// TIA Portal project "FactoryIO_assembler" (V19)
// Vorlageprojekt für das Buch mit Zielsystem S7-1200

(* hardware
DEVICE "S7-1200-Station_1"  S7-1200 Station
   slot 0: "Baugruppenträger_0"  Rack  V1.0
   slot 1: "PLC_1"  CPU 1211C DC/DC/DC  6ES7 211-1AE40-0XB0  V4.1
*)

// ===== PLC "PLC_1"  CPU 1211C DC/DC/DC =====

VAR_GLOBAL   // PLC tag table "Standard-Variablentabelle"
   "Move_X" AT %A0.0 : Bool;
   "Moving_X" AT %E0.0 : Bool;
   "Moving_Z" AT %E0.1 : Bool;
   "FactoryIO_Running" AT %I1.7 : Bool;
   "Start" AT %I1.2 : Bool;
   "Reset" AT %I1.3 : Bool;
   "Stop" AT %I1.4 : Bool;
   "Emergency_Stop" AT %I1.5 : Bool;
   "Auto" AT %I1.6 : Bool;
   "Move_Z" AT %Q0.1 : Bool;
   "Grab" AT %Q0.2 : Bool;
   "Lids_conveyor" AT %Q0.3 : Bool;
   "Clamp_lid" AT %Q0.4 : Bool;
   "Pos_raise" AT %Q0.5 : Bool;
   "Bases_conveyor" AT %Q0.6 : Bool;
   "Start_light" AT %Q1.1 : Bool;
   "Reset light" AT %Q1.2 : Bool;
   "Stop light" AT %Q1.3 : Bool;
   "Counter" AT %QD30 : DInt;
   "Item_detected" AT %I0.2 : Bool;
   "Lid_at_place" AT %I0.3 : Bool;
   "Lid_clamped" AT %I0.4 : Bool;
   "Pos_at_limit (lids)" AT %I0.5 : Bool;
   "Base_at_place" AT %I0.6 : Bool;
   "Base_clamped" AT %I0.7 : Bool;
   "Pos_at_limit (bases)" AT %I1.0 : Bool;
   "Part_leaving" AT %I1.1 : Bool;
   "Clamp_base" AT %Q0.7 : Bool;
   "Pos_raise (bases)" AT %Q1.0 : Bool;
   "Tag_1" AT %M0.0 : Bool;
   "Tag_2" AT %M0.1 : Bool;
   "Tag_3" AT %M0.2 : Bool;
   "Tag_4" AT %M0.3 : Bool;
   "Tag_5" AT %M0.4 : Bool;
   "Tag_6" AT %M0.5 : Bool;
   "Lid_aligned" AT %M0.6 : Bool;
   "Tag_7" AT %M0.7 : Bool;
   "Tag_8" AT %M1.0 : Bool;
   "base_aligned" AT %M1.1 : Bool;
   "Tag_9" AT %M1.2 : Bool;
   "Move_Z_bit" AT %M1.3 : Bool;
   "Tag_10" AT %M1.4 : Bool;
   "Tag_11" AT %M1.5 : Bool;
   "Tag_12" AT %M1.6 : Bool;
   "Tag_13" AT %M1.7 : Bool;
   "Tag_14" AT %M2.0 : Bool;
   "Tag_15" AT %M2.2 : Bool;
   "Move_Z_bit2" AT %M2.1 : Bool;
   "combined_bit" AT %M2.3 : Bool;
   "Tag_16" AT %M2.4 : Bool;
   "Home_bit" AT %M2.5 : Bool;
   "Tag_17" AT %M2.6 : Bool;
END_VAR

// folder: System blocks/Program resources

DATA_BLOCK "IEC_Timer_0_DB"   // DB1
{ S7_Optimized_Access := 'TRUE' }
AUTHOR : Simatic
FAMILY : IEC
NAME : IEC_TMR
VERSION : 1.0
// stored: InstanceOfName IEC_TIMER
"IEC_TIMER"
BEGIN
END_DATA_BLOCK

DATA_BLOCK "IEC_Timer_0_DB_1"   // DB2
{ S7_Optimized_Access := 'TRUE' }
AUTHOR : Simatic
FAMILY : IEC
NAME : IEC_TMR
VERSION : 1.0
// stored: InstanceOfName IEC_TIMER
"IEC_TIMER"
BEGIN
END_DATA_BLOCK

DATA_BLOCK "IEC_Timer_0_DB_2"   // DB3
{ S7_Optimized_Access := 'TRUE' }
AUTHOR : Simatic
FAMILY : IEC
NAME : IEC_TMR
VERSION : 1.0
// stored: InstanceOfName IEC_TIMER
"IEC_TIMER"
BEGIN
END_DATA_BLOCK

// folder: (top level)

FUNCTION "conveyor" : Void   // FC1, LAD
{ S7_Optimized_Access := 'TRUE' }
VERSION : 0.1
   VAR_TEMP   // added for the SCL form of the ladder/FBD networks
      _w1 : Bool;
   END_VAR
BEGIN

REGION Network 1
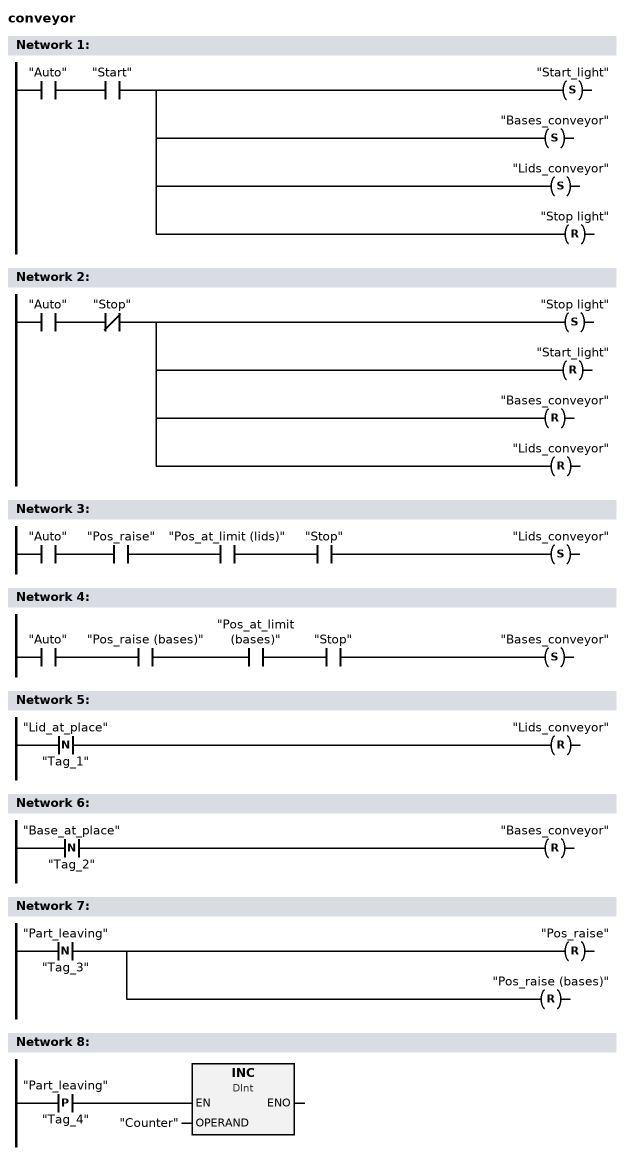
   RUNG wire#powerrail
      Contact( "Auto" )
      Contact( "Start" )
      wire#w1
      S_Coil( "Start_light" )
   END_RUNG
   RUNG wire#w1
      S_Coil( "Bases_conveyor" )
   END_RUNG
   RUNG wire#w1
      S_Coil( "Lids_conveyor" )
   END_RUNG
   RUNG wire#w1
      R_Coil( "Stop light" )
   END_RUNG
   // the same network as SCL:
   IF "Auto" AND "Start" THEN
       "Start_light" := TRUE;
       "Bases_conveyor" := TRUE;
       "Lids_conveyor" := TRUE;
       "Stop light" := FALSE;
   END_IF;
END_REGION

REGION Network 2
   RUNG wire#powerrail
      Contact( "Auto" )
      I_Contact( "Stop" )
      wire#w1
      S_Coil( "Stop light" )
   END_RUNG
   RUNG wire#w1
      R_Coil( "Start_light" )
   END_RUNG
   RUNG wire#w1
      R_Coil( "Bases_conveyor" )
   END_RUNG
   RUNG wire#w1
      R_Coil( "Lids_conveyor" )
   END_RUNG
   // the same network as SCL:
   IF "Auto" AND NOT "Stop" THEN
       "Stop light" := TRUE;
       "Start_light" := FALSE;
       "Bases_conveyor" := FALSE;
       "Lids_conveyor" := FALSE;
   END_IF;
END_REGION

REGION Network 3
   RUNG wire#powerrail
      Contact( "Auto" )
      Contact( "Pos_raise" )
      Contact( "Pos_at_limit (lids)" )
      Contact( "Stop" )
      S_Coil( "Lids_conveyor" )
   END_RUNG
   // the same network as SCL:
   IF "Auto" AND "Pos_raise" AND "Pos_at_limit (lids)" AND "Stop" THEN "Lids_conveyor" := TRUE; END_IF;
END_REGION

REGION Network 4
   RUNG wire#powerrail
      Contact( "Auto" )
      Contact( "Pos_raise (bases)" )
      Contact( "Pos_at_limit (bases)" )
      Contact( "Stop" )
      S_Coil( "Bases_conveyor" )
   END_RUNG
   // the same network as SCL:
   IF "Auto" AND "Pos_raise (bases)" AND "Pos_at_limit (bases)" AND "Stop" THEN
       "Bases_conveyor" := TRUE;
   END_IF;
END_REGION

REGION Network 5
   RUNG wire#powerrail
      N_Contact(operand := "Lid_at_place", bit := "Tag_1")
      R_Coil( "Lids_conveyor" )
   END_RUNG
   // the same network as SCL:
   #_w1 := NOT "Lid_at_place" AND "Tag_1";   // falling edge of "Lid_at_place"
   "Tag_1" := "Lid_at_place";
   IF #_w1 THEN "Lids_conveyor" := FALSE; END_IF;
END_REGION

REGION Network 6
   RUNG wire#powerrail
      N_Contact(operand := "Base_at_place", bit := "Tag_2")
      R_Coil( "Bases_conveyor" )
   END_RUNG
   // the same network as SCL:
   #_w1 := NOT "Base_at_place" AND "Tag_2";   // falling edge of "Base_at_place"
   "Tag_2" := "Base_at_place";
   IF #_w1 THEN "Bases_conveyor" := FALSE; END_IF;
END_REGION

REGION Network 7
   RUNG wire#powerrail
      N_Contact(operand := "Part_leaving", bit := "Tag_3")
      wire#w1
      R_Coil( "Pos_raise" )
   END_RUNG
   RUNG wire#w1
      R_Coil( "Pos_raise (bases)" )
   END_RUNG
   // the same network as SCL:
   #_w1 := NOT "Part_leaving" AND "Tag_3";   // falling edge of "Part_leaving"
   "Tag_3" := "Part_leaving";
   IF #_w1 THEN
       "Pos_raise" := FALSE;
       "Pos_raise (bases)" := FALSE;
   END_IF;
END_REGION

REGION Network 8
   RUNG wire#powerrail
      P_Contact(operand := "Part_leaving", bit := "Tag_4")
      { S7_Templates := "DestType := DInt" } Inc( "Counter" )
   END_RUNG
   // the same network as SCL:
   #_w1 := "Part_leaving" AND NOT "Tag_4";   // rising edge of "Part_leaving"
   "Tag_4" := "Part_leaving";
   IF #_w1 THEN "Counter" := "Counter" + 1; END_IF;
END_REGION
END_FUNCTION

FUNCTION "clamp" : Void   // FC2, LAD
{ S7_Optimized_Access := 'TRUE' }
VERSION : 0.1
   VAR_TEMP   // added for the SCL form of the ladder/FBD networks
      _w1 : Bool;
   END_VAR
BEGIN

REGION Network 1
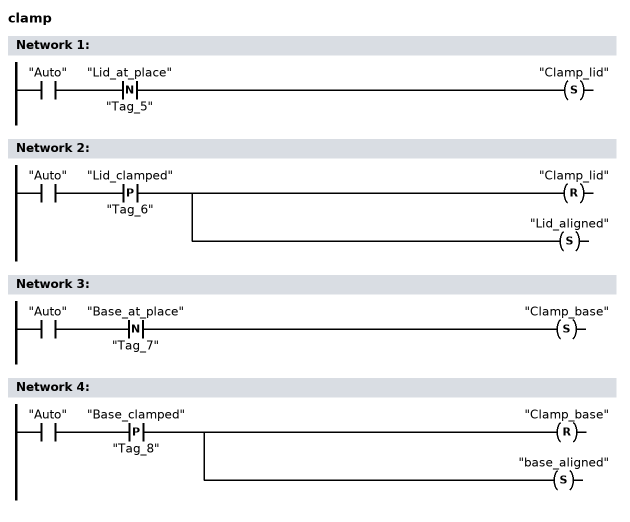
   RUNG wire#powerrail
      Contact( "Auto" )
      N_Contact(operand := "Lid_at_place", bit := "Tag_5")
      S_Coil( "Clamp_lid" )
   END_RUNG
   // the same network as SCL:
   #_w1 := "Auto" AND NOT "Lid_at_place" AND "Tag_5";   // falling edge of "Lid_at_place"
   "Tag_5" := "Lid_at_place";
   IF #_w1 THEN "Clamp_lid" := TRUE; END_IF;
END_REGION

REGION Network 2
   RUNG wire#powerrail
      Contact( "Auto" )
      P_Contact(operand := "Lid_clamped", bit := "Tag_6")
      wire#w1
      R_Coil( "Clamp_lid" )
   END_RUNG
   RUNG wire#w1
      S_Coil( "Lid_aligned" )
   END_RUNG
   // the same network as SCL:
   #_w1 := "Auto" AND "Lid_clamped" AND NOT "Tag_6";   // rising edge of "Lid_clamped"
   "Tag_6" := "Lid_clamped";
   IF #_w1 THEN
       "Clamp_lid" := FALSE;
       "Lid_aligned" := TRUE;
   END_IF;
END_REGION

REGION Network 3
   RUNG wire#powerrail
      Contact( "Auto" )
      N_Contact(operand := "Base_at_place", bit := "Tag_7")
      S_Coil( "Clamp_base" )
   END_RUNG
   // the same network as SCL:
   #_w1 := "Auto" AND NOT "Base_at_place" AND "Tag_7";   // falling edge of "Base_at_place"
   "Tag_7" := "Base_at_place";
   IF #_w1 THEN "Clamp_base" := TRUE; END_IF;
END_REGION

REGION Network 4
   RUNG wire#powerrail
      Contact( "Auto" )
      P_Contact(operand := "Base_clamped", bit := "Tag_8")
      wire#w1
      R_Coil( "Clamp_base" )
   END_RUNG
   RUNG wire#w1
      S_Coil( "base_aligned" )
   END_RUNG
   // the same network as SCL:
   #_w1 := "Auto" AND "Base_clamped" AND NOT "Tag_8";   // rising edge of "Base_clamped"
   "Tag_8" := "Base_clamped";
   IF #_w1 THEN
       "Clamp_base" := FALSE;
       "base_aligned" := TRUE;
   END_IF;
END_REGION
END_FUNCTION

FUNCTION "pick_and_place" : Void   // FC3, LAD
{ S7_Optimized_Access := 'TRUE' }
VERSION : 0.1
   VAR_TEMP   // added for the SCL form of the ladder/FBD networks
      _w1 : Bool;
   END_VAR
BEGIN

REGION Network 1
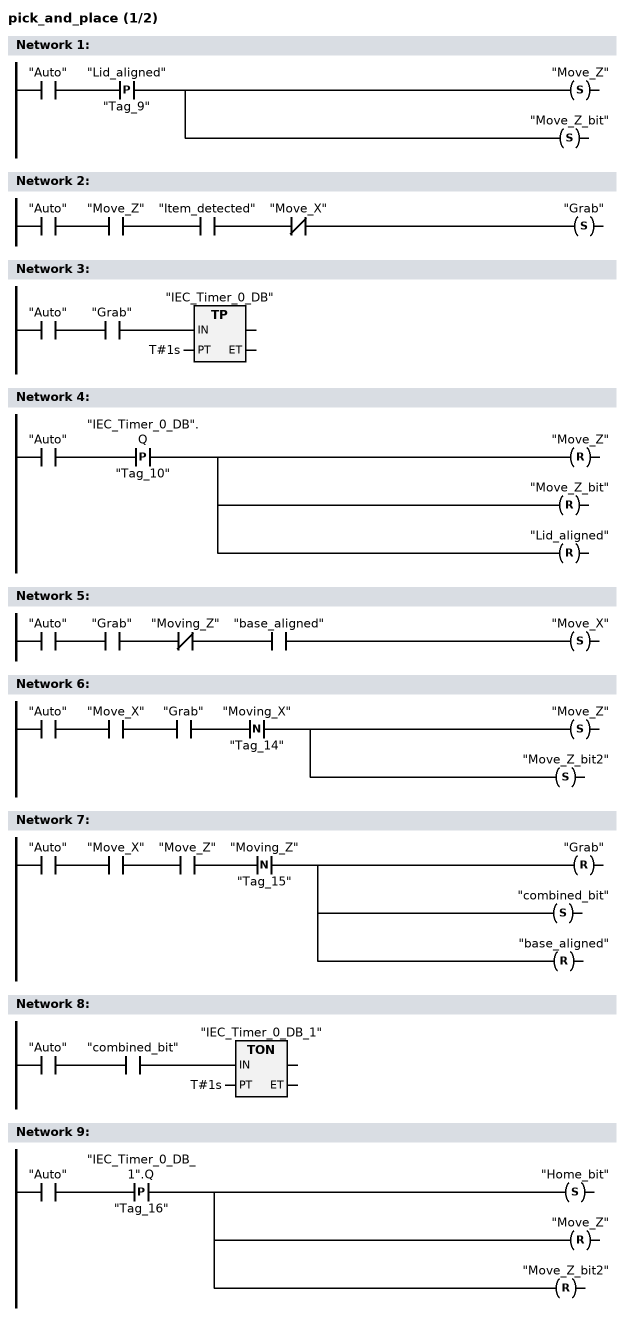
   RUNG wire#powerrail
      Contact( "Auto" )
      P_Contact(operand := "Lid_aligned", bit := "Tag_9")
      wire#w1
      S_Coil( "Move_Z" )
   END_RUNG
   RUNG wire#w1
      S_Coil( "Move_Z_bit" )
   END_RUNG
   // the same network as SCL:
   #_w1 := "Auto" AND "Lid_aligned" AND NOT "Tag_9";   // rising edge of "Lid_aligned"
   "Tag_9" := "Lid_aligned";
   IF #_w1 THEN
       "Move_Z" := TRUE;
       "Move_Z_bit" := TRUE;
   END_IF;
END_REGION

REGION Network 2
   RUNG wire#powerrail
      Contact( "Auto" )
      Contact( "Move_Z" )
      Contact( "Item_detected" )
      I_Contact( "Move_X" )
      S_Coil( "Grab" )
   END_RUNG
   // the same network as SCL:
   IF "Auto" AND "Move_Z" AND "Item_detected" AND NOT "Move_X" THEN "Grab" := TRUE; END_IF;
END_REGION

REGION Network 3
   "IEC_Timer_0_DB".TP(IN := "Auto" AND "Grab", PT := T#1s);
END_REGION

REGION Network 4
   RUNG wire#powerrail
      Contact( "Auto" )
      P_Contact(operand := "IEC_Timer_0_DB".Q, bit := "Tag_10")
      wire#w1
      R_Coil( "Move_Z" )
   END_RUNG
   RUNG wire#w1
      R_Coil( "Move_Z_bit" )
   END_RUNG
   RUNG wire#w1
      R_Coil( "Lid_aligned" )
   END_RUNG
   // the same network as SCL:
   #_w1 := "Auto" AND "IEC_Timer_0_DB".Q AND NOT "Tag_10";   // rising edge of "IEC_Timer_0_DB".Q
   "Tag_10" := "IEC_Timer_0_DB".Q;
   IF #_w1 THEN
       "Move_Z" := FALSE;
       "Move_Z_bit" := FALSE;
       "Lid_aligned" := FALSE;
   END_IF;
END_REGION

REGION Network 5
   RUNG wire#powerrail
      Contact( "Auto" )
      Contact( "Grab" )
      I_Contact( "Moving_Z" )
      Contact( "base_aligned" )
      S_Coil( "Move_X" )
   END_RUNG
   // the same network as SCL:
   IF "Auto" AND "Grab" AND NOT "Moving_Z" AND "base_aligned" THEN "Move_X" := TRUE; END_IF;
END_REGION

REGION Network 6
   RUNG wire#powerrail
      Contact( "Auto" )
      Contact( "Move_X" )
      Contact( "Grab" )
      N_Contact(operand := "Moving_X", bit := "Tag_14")
      wire#w1
      S_Coil( "Move_Z" )
   END_RUNG
   RUNG wire#w1
      S_Coil( "Move_Z_bit2" )
   END_RUNG
   // the same network as SCL:
   #_w1 := "Auto" AND "Move_X" AND "Grab" AND NOT "Moving_X" AND "Tag_14";   // falling edge of "Moving_X"
   "Tag_14" := "Moving_X";
   IF #_w1 THEN
       "Move_Z" := TRUE;
       "Move_Z_bit2" := TRUE;
   END_IF;
END_REGION

REGION Network 7
   RUNG wire#powerrail
      Contact( "Auto" )
      Contact( "Move_X" )
      Contact( "Move_Z" )
      N_Contact(operand := "Moving_Z", bit := "Tag_15")
      wire#w1
      R_Coil( "Grab" )
   END_RUNG
   RUNG wire#w1
      S_Coil( "combined_bit" )
   END_RUNG
   RUNG wire#w1
      R_Coil( "base_aligned" )
   END_RUNG
   // the same network as SCL:
   #_w1 := "Auto" AND "Move_X" AND "Move_Z" AND NOT "Moving_Z" AND "Tag_15";   // falling edge of "Moving_Z"
   "Tag_15" := "Moving_Z";
   IF #_w1 THEN
       "Grab" := FALSE;
       "combined_bit" := TRUE;
       "base_aligned" := FALSE;
   END_IF;
END_REGION

REGION Network 8
   "IEC_Timer_0_DB_1".TON(IN := "Auto" AND "combined_bit", PT := T#1s);
END_REGION

REGION Network 9
   RUNG wire#powerrail
      Contact( "Auto" )
      P_Contact(operand := "IEC_Timer_0_DB_1".Q, bit := "Tag_16")
      wire#w1
      S_Coil( "Home_bit" )
   END_RUNG
   RUNG wire#w1
      R_Coil( "Move_Z" )
   END_RUNG
   RUNG wire#w1
      R_Coil( "Move_Z_bit2" )
   END_RUNG
   // the same network as SCL:
   #_w1 := "Auto" AND "IEC_Timer_0_DB_1".Q AND NOT "Tag_16";   // rising edge of "IEC_Timer_0_DB_1".Q
   "Tag_16" := "IEC_Timer_0_DB_1".Q;
   IF #_w1 THEN
       "Home_bit" := TRUE;
       "Move_Z" := FALSE;
       "Move_Z_bit2" := FALSE;
   END_IF;
END_REGION

REGION Network 10
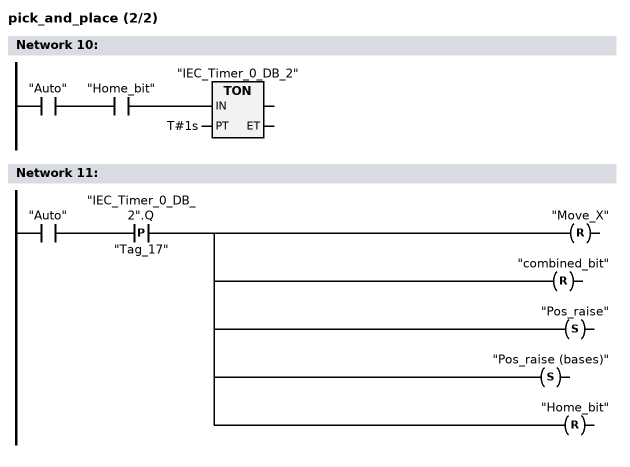
   "IEC_Timer_0_DB_2".TON(IN := "Auto" AND "Home_bit", PT := T#1s);
END_REGION

REGION Network 11
   RUNG wire#powerrail
      Contact( "Auto" )
      P_Contact(operand := "IEC_Timer_0_DB_2".Q, bit := "Tag_17")
      wire#w1
      R_Coil( "Move_X" )
   END_RUNG
   RUNG wire#w1
      R_Coil( "combined_bit" )
   END_RUNG
   RUNG wire#w1
      S_Coil( "Pos_raise" )
   END_RUNG
   RUNG wire#w1
      S_Coil( "Pos_raise (bases)" )
   END_RUNG
   RUNG wire#w1
      R_Coil( "Home_bit" )
   END_RUNG
   // the same network as SCL:
   #_w1 := "Auto" AND "IEC_Timer_0_DB_2".Q AND NOT "Tag_17";   // rising edge of "IEC_Timer_0_DB_2".Q
   "Tag_17" := "IEC_Timer_0_DB_2".Q;
   IF #_w1 THEN
       "Move_X" := FALSE;
       "combined_bit" := FALSE;
       "Pos_raise" := TRUE;
       "Pos_raise (bases)" := TRUE;
       "Home_bit" := FALSE;
   END_IF;
END_REGION
END_FUNCTION

FUNCTION "MHJ-PLC-Lab-Function-S71200" : Void   // FC9000, SCL
{ S7_Optimized_Access := 'TRUE' }
VERSION : 0.1
   VAR_TEMP
      rdTimeReturn : Int;
      outputTime : DTL;
      SyncVal : Byte;
      forVal : Int;
      forVal_2 : Int;
      Value : Byte;
   END_VAR
   VAR CONSTANT
      CompVal : Byte := 16#34;
      Value_01 : Byte := 16#11;
      Value_01_DW : DWord := 16#A165_D992;
      Value_02_DW : DWord := 16#58BE_4401;
   END_VAR
BEGIN

   #Value:=PEEK(area := 16#82,
        dbNumber := 0,
        byteOffset := 511);
   #Value := #Value + 1;

   POKE(area := 16#82,
        dbNumber := 0,
        byteOffset := 511,
        value := #Value);

   POKE(area:=16#81,
        dbNumber:=0,
        byteOffset:=1016,
        value:=#Value_01_DW);
   POKE(area := 16#81,
        dbNumber := 0,
        byteOffset := 1020,
        value := #Value_02_DW);

   POKE(area := 16#81,
        dbNumber := 0,
        byteOffset := 511,
        value := B#16#00);

   FOR #forVal := 0 TO 120 DO
       FOR #forVal_2:=0 TO 10 DO
           #rdTimeReturn:=RD_SYS_T(#outputTime);
           #rdTimeReturn := WR_SYS_T(#outputTime);
           #rdTimeReturn := RD_SYS_T(#outputTime);
           #rdTimeReturn := WR_SYS_T(#outputTime);
       END_FOR;
       #SyncVal:= PEEK(area := 16#81,
                      dbNumber := 0,
                      byteOffset := 511);
       IF #SyncVal = #CompVal THEN
          GOTO M_1;
       END_IF;
   END_FOR;
   RETURN;

   M_1:
   POKE(area := 16#81,
        dbNumber := 0,
        byteOffset := 511,
        value := B#16#0);
END_FUNCTION

ORGANIZATION_BLOCK "Main"   // OB1, FBD, ProgramCycle
TITLE = "Main Program Sweep (Cycle)"
{ S7_Optimized_Access := 'TRUE' }
VERSION : 0.1
   VAR_INPUT
      Initial_Call : Bool;   // Initial call of this OB
      Remanence : Bool;   // =True, if remanent data are available
   END_VAR
BEGIN

REGION Network 1: Konnektierungsbaustein für PLC-Lab
   // Im Netzwerk 1 wird der Konnektierungsbaustein für PLC-Lab aufgerufen.
   // Dieser Aufruf darf nicht entfernt werden!
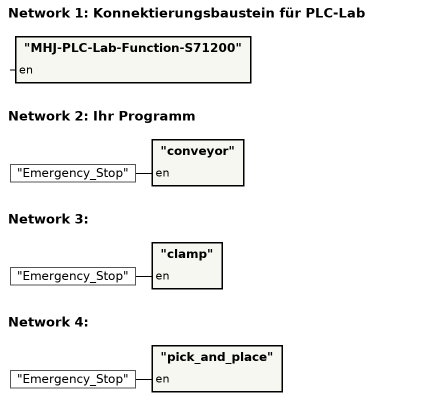
   "MHJ-PLC-Lab-Function-S71200"();
END_REGION

REGION Network 2: Ihr Programm
   // Schreiben Sie ab Netzwerk 2 Ihr Programm
   IF "Emergency_Stop" THEN "conveyor"(); END_IF;
END_REGION

REGION Network 3
   IF "Emergency_Stop" THEN "clamp"(); END_IF;
END_REGION

REGION Network 4
   IF "Emergency_Stop" THEN "pick_and_place"(); END_IF;
END_REGION
END_ORGANIZATION_BLOCK